// TwinCAT 3 PLC project TestPlcProject
// Title: TestPlcProject
// Company: TestPlcProject
// ProjectVersion: 0.1.0
// ProgramVersion: 3.1.4023.0
// libraries:
//   Tc2_Standard, * (Beckhoff Automation GmbH)
//   Tc2_System, * (Beckhoff Automation GmbH)
//   Tc3_Module, * (Beckhoff Automation GmbH)
// project tree:
//   / PlcTask.TcTTO (not stored)
//   POUs/ FB_TestFb1.TcPOU, MAIN.TcPOU

// ---- POUs/FB_TestFb1.TcPOU
FUNCTION_BLOCK FB_TestFb1
VAR_INPUT
END_VAR
VAR_OUTPUT
END_VAR
VAR
END_VAR

END_FUNCTION_BLOCK

// ---- POUs/MAIN.TcPOU
PROGRAM MAIN
VAR
END_VAR

END_PROGRAM
